// Mitsubishi GX Works2 project: TESTES   PLC: Q03UDV
// LRI_2023

PROGRAM MAIN
VAR
  yo : INT;
  TS0 : BOOL;
  RT0 : BOOL;
END_VAR
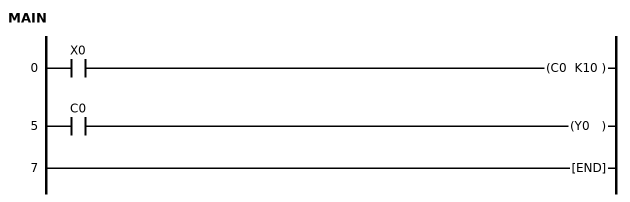
0     LD      X0
      OUT     C0 K10
5     LD      C0
      OUT     Y0
7     END
END_PROGRAM
